PROGRAM MAIN
VAR
END_VAR

PRG_DIAGNOSTIC();
PRG_SXR_VAC();

END_PROGRAM

(* stored: Version 1.1.0.1, ProductVersion 3.1.4022.16
   POU MAIN: Id {514fb895-bcbe-4717-9c32-df3e61678814}, SpecialFunc None *)
